TYPE T_HTTP_URL : STRING(GVL_HTTP_PARAMETERS.MAX_HTTP_URL_LENGTH); END_TYPE

(* stored: Version 1.1.0.1, ProductVersion 3.1.4020.3
   DUT T_HTTP_URL: Id {45ff549d-ffdf-4b30-9a35-a35e287c6f47} *)
